{attribute 'strict'}
TYPE E_CS_Status :
(
    Offline := 0,
	Idle,
	DriveReady,
    ReadyToWork,
    Pou_Runing,
    Pou_Run_Pause,
    Pou_Run_Down,
	EStop,
    Error,
	LessHome,
	StopMess,
	LocalControl,
	DriverOn
);
END_TYPE

(* stored: Version 1.1.0.1, ProductVersion 3.1.4024.16
   DUT E_CS_Status: Id {d7ecf668-c873-4ad4-b273-fa44e78bd863} *)
